{attribute 'qualified_only'}
{attribute 'strict'}
{attribute 'to_string'}
TYPE E_CommandPriority :
(
	LOW := 0,
  NORMAL,
  HIGH
);
END_TYPE

(* stored: Version 1.1.0.1
   DUT E_CommandPriority: Id {31fcbffd-c546-442b-9084-71191a16afee} *)
